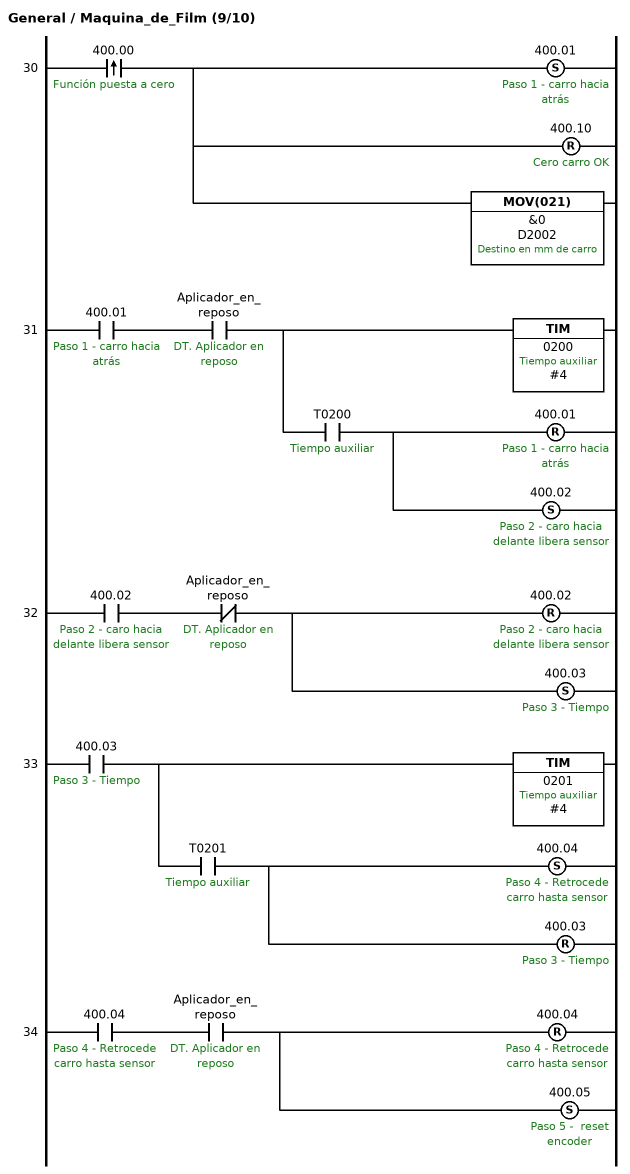
; [picture p24: General / Maquina_de_Film, rungs 30-34]
; rung 30
@LD 400.00  ; Función puesta a cero
SET 400.01  ; Paso 1 - carro hacia atrás
RSET 400.10  ; Cero carro OK
MOV(021) &0 D2002  ; Destino en mm de carro
; rung 31
LD 400.01  ; Paso 1 - carro hacia atrás
AND Aplicador_en_reposo  ; DT. Aplicador en reposo
TIM 0200 #4  ; Tiempo auxiliar
AND T0200  ; Tiempo auxiliar
RSET 400.01  ; Paso 1 - carro hacia atrás
SET 400.02  ; Paso 2 - caro hacia delante libera sensor
; rung 32
LD 400.02  ; Paso 2 - caro hacia delante libera sensor
ANDNOT Aplicador_en_reposo  ; DT. Aplicador en reposo
RSET 400.02  ; Paso 2 - caro hacia delante libera sensor
SET 400.03  ; Paso 3 - Tiempo
; rung 33
LD 400.03  ; Paso 3 - Tiempo
TIM 0201 #4  ; Tiempo auxiliar
AND T0201  ; Tiempo auxiliar
SET 400.04  ; Paso 4 - Retrocede carro hasta sensor
RSET 400.03  ; Paso 3 - Tiempo
; rung 34
LD 400.04  ; Paso 4 - Retrocede carro hasta sensor
AND Aplicador_en_reposo  ; DT. Aplicador en reposo
RSET 400.04  ; Paso 4 - Retrocede carro hasta sensor
SET 400.05  ; Paso 5 -  reset encoder

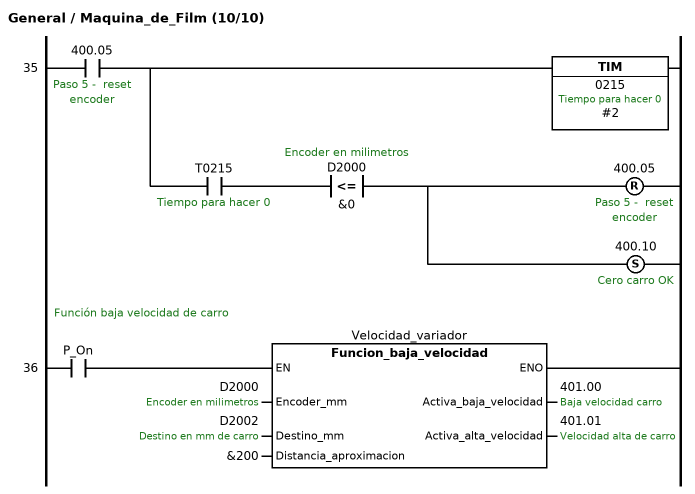
; rung 35
LD 400.05  ; Paso 5 -  reset encoder
TIM 0215 #2  ; Tiempo para hacer 0
AND T0215  ; Tiempo para hacer 0
AND<=SL(318) D2000 &0  ; Encoder en milimetros
RSET 400.05  ; Paso 5 -  reset encoder
SET 400.10  ; Cero carro OK
; rung 36: Función baja velocidad de carro
LD P_On
CALL Velocidad_variador : Funcion_baja_velocidad (Encoder_mm := D2000, Destino_mm := D2002, Distancia_aproximacion := &200, Activa_baja_velocidad => 401.00, Activa_alta_velocidad => 401.01)  ; Encoder en milimetros, Destino en mm de carro, Baja velocidad carro, Velocidad alta de carro

### Section Compuerta

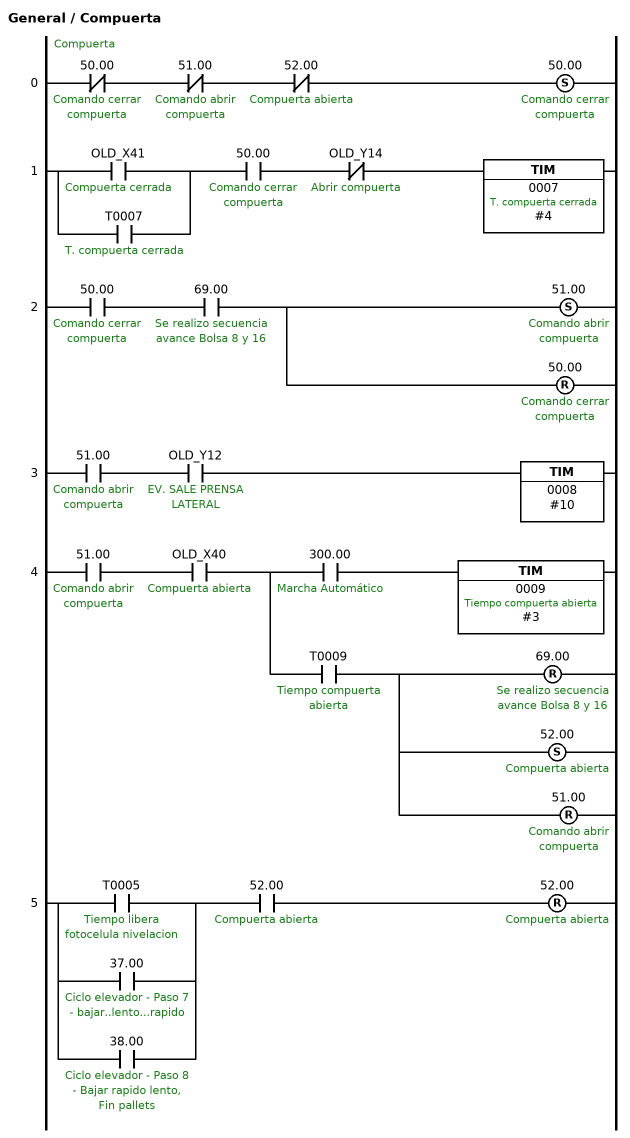
; rung 0: Compuerta
LDNOT 50.00  ; Comando cerrar compuerta
ANDNOT 51.00  ; Comando abrir compuerta
ANDNOT 52.00  ; Compuerta abierta
SET 50.00  ; Comando cerrar compuerta
; rung 1
LD OLD_X41  ; Compuerta cerrada
OR T0007  ; T. compuerta cerrada
AND 50.00  ; Comando cerrar compuerta
ANDNOT OLD_Y14  ; Abrir compuerta
TIM 0007 #4  ; T. compuerta cerrada
; rung 2
LD 50.00  ; Comando cerrar compuerta
AND 69.00  ; Se realizo secuencia avance Bolsa 8 y 16
SET 51.00  ; Comando abrir compuerta
RSET 50.00  ; Comando cerrar compuerta
; rung 3
LD 51.00  ; Comando abrir compuerta
AND OLD_Y12  ; EV. SALE PRENSA LATERAL
TIM 0008 #10
; rung 4
LD 51.00  ; Comando abrir compuerta
AND OLD_X40  ; Compuerta abierta
OUT TR0
AND 300.00  ; Marcha Automático
TIM 0009 #3  ; Tiempo compuerta abierta
LD TR0
AND T0009  ; Tiempo compuerta abierta
RSET 69.00  ; Se realizo secuencia avance Bolsa 8 y 16
SET 52.00  ; Compuerta abierta
RSET 51.00  ; Comando abrir compuerta
; rung 5
LD T0005  ; Tiempo libera fotocelula nivelacion
OR 37.00  ; Ciclo elevador - Paso 7 - bajar..lento...rapido
OR 38.00  ; Ciclo elevador - Paso 8 - Bajar rapido lento, Fin pallets
AND 52.00  ; Compuerta abierta
RSET 52.00  ; Compuerta abierta

### Section Carro_pala

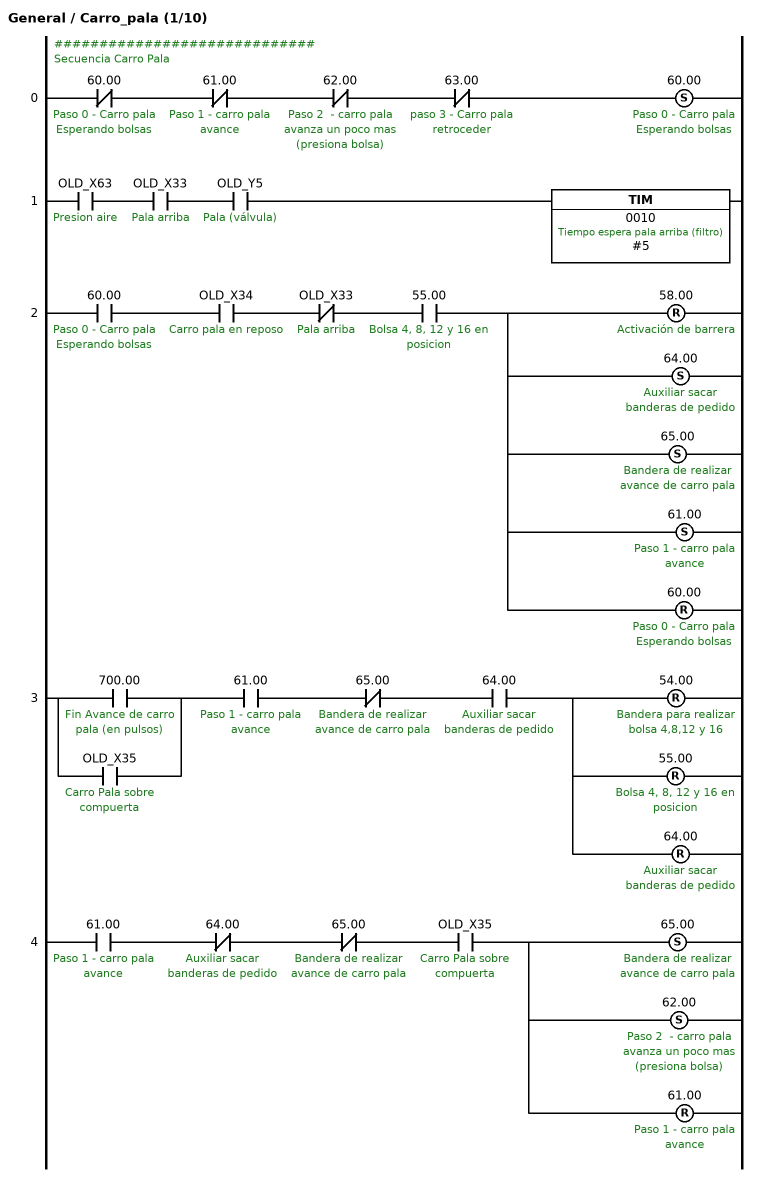
; rung 0: ############################# / Secuencia Carro Pala
LDNOT 60.00  ; Paso 0 - Carro pala Esperando bolsas
ANDNOT 61.00  ; Paso 1 - carro pala avance
ANDNOT 62.00  ; Paso 2  - carro pala avanza un poco mas (presiona bolsa)
ANDNOT 63.00  ; paso 3 - Carro pala retroceder
SET 60.00  ; Paso 0 - Carro pala Esperando bolsas
; rung 1
LD OLD_X63  ; Presion aire
AND OLD_X33  ; Pala arriba
AND OLD_Y5  ; Pala (válvula)
TIM 0010 #5  ; Tiempo espera pala arriba (filtro)
; rung 2
LD 60.00  ; Paso 0 - Carro pala Esperando bolsas
AND OLD_X34  ; Carro pala en reposo
ANDNOT OLD_X33  ; Pala arriba
AND 55.00  ; Bolsa 4, 8, 12 y 16 en posicion
RSET 58.00  ; Activación de barrera
SET 64.00  ; Auxiliar sacar banderas de pedido
SET 65.00  ; Bandera de realizar avance de carro pala
SET 61.00  ; Paso 1 - carro pala avance
RSET 60.00  ; Paso 0 - Carro pala Esperando bolsas
; rung 3
LD 700.00  ; Fin Avance de carro pala (en pulsos)
OR OLD_X35  ; Carro Pala sobre compuerta
AND 61.00  ; Paso 1 - carro pala avance
ANDNOT 65.00  ; Bandera de realizar avance de carro pala
AND 64.00  ; Auxiliar sacar banderas de pedido
RSET 54.00  ; Bandera para realizar bolsa 4,8,12 y 16
RSET 55.00  ; Bolsa 4, 8, 12 y 16 en posicion
RSET 64.00  ; Auxiliar sacar banderas de pedido
; rung 4
LD 61.00  ; Paso 1 - carro pala avance
ANDNOT 64.00  ; Auxiliar sacar banderas de pedido
ANDNOT 65.00  ; Bandera de realizar avance de carro pala
AND OLD_X35  ; Carro Pala sobre compuerta
SET 65.00  ; Bandera de realizar avance de carro pala
SET 62.00  ; Paso 2  - carro pala avanza un poco mas (presiona bolsa)
RSET 61.00  ; Paso 1 - carro pala avance

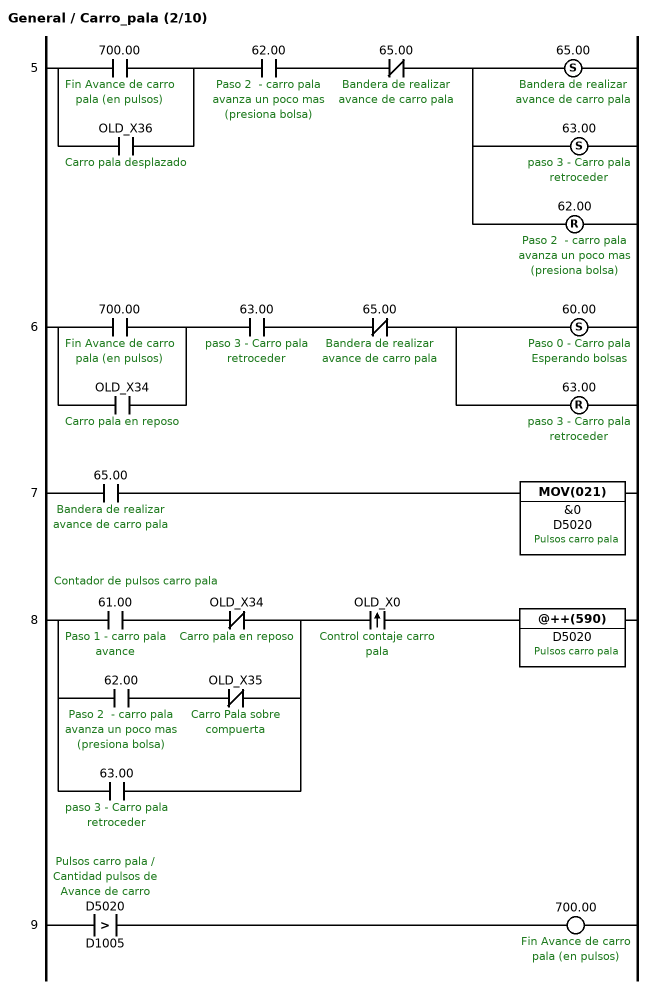
; rung 5
LD 700.00  ; Fin Avance de carro pala (en pulsos)
OR OLD_X36  ; Carro pala desplazado
AND 62.00  ; Paso 2  - carro pala avanza un poco mas (presiona bolsa)
ANDNOT 65.00  ; Bandera de realizar avance de carro pala
SET 65.00  ; Bandera de realizar avance de carro pala
SET 63.00  ; paso 3 - Carro pala retroceder
RSET 62.00  ; Paso 2  - carro pala avanza un poco mas (presiona bolsa)
; rung 6
LD 700.00  ; Fin Avance de carro pala (en pulsos)
OR OLD_X34  ; Carro pala en reposo
AND 63.00  ; paso 3 - Carro pala retroceder
ANDNOT 65.00  ; Bandera de realizar avance de carro pala
SET 60.00  ; Paso 0 - Carro pala Esperando bolsas
RSET 63.00  ; paso 3 - Carro pala retroceder
; rung 7
LD 65.00  ; Bandera de realizar avance de carro pala
MOV(021) &0 D5020  ; Pulsos carro pala
; rung 8: Contador de pulsos carro pala
LD 61.00  ; Paso 1 - carro pala avance
ANDNOT OLD_X34  ; Carro pala en reposo
LD 62.00  ; Paso 2  - carro pala avanza un poco mas (presiona bolsa)
ANDNOT OLD_X35  ; Carro Pala sobre compuerta
ORLD
OR 63.00  ; paso 3 - Carro pala retroceder
@AND OLD_X0  ; Control contaje carro pala
@++(590) D5020  ; Pulsos carro pala
; rung 9
LD>(320) D5020 D1005  ; Pulsos carro pala, Cantidad pulsos de Avance de carro
OUT 700.00  ; Fin Avance de carro pala (en pulsos)

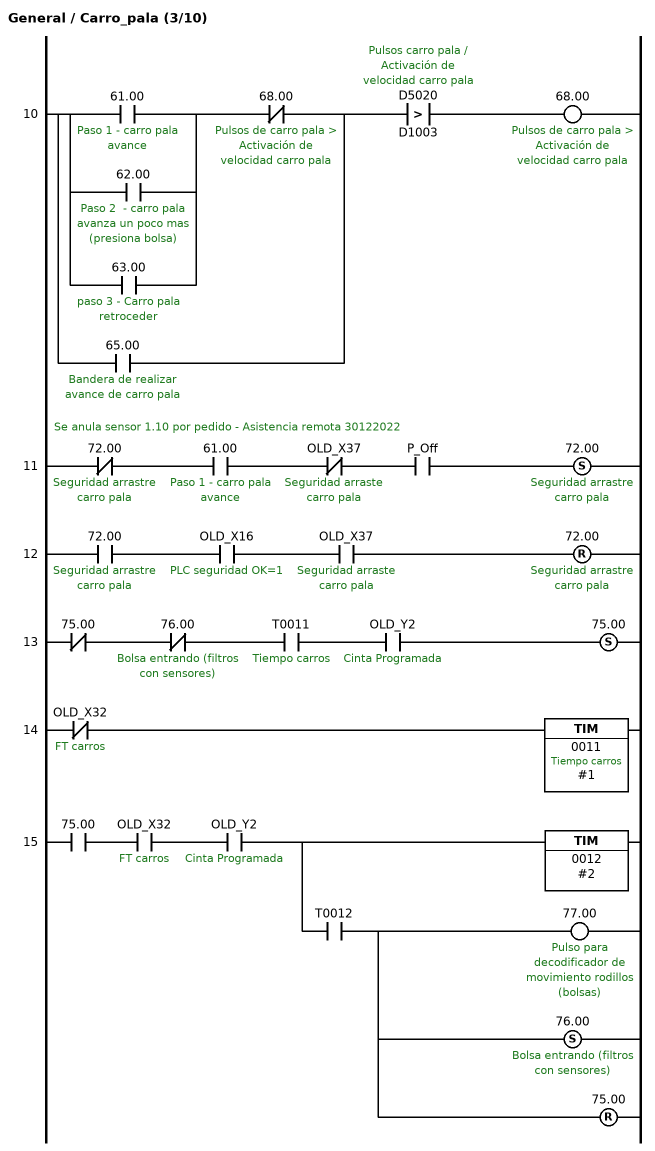
; rung 10
LD 61.00  ; Paso 1 - carro pala avance
OR 62.00  ; Paso 2  - carro pala avanza un poco mas (presiona bolsa)
OR 63.00  ; paso 3 - Carro pala retroceder
ANDNOT 68.00  ; Pulsos de carro pala > Activación de velocidad carro pala
OR 65.00  ; Bandera de realizar avance de carro pala
AND>L(321) D5020 D1003  ; Pulsos carro pala, Activación de velocidad carro pala
OUT 68.00  ; Pulsos de carro pala > Activación de velocidad carro pala
; rung 11: Se anula sensor 1.10 por pedido - Asistencia remota 30122022
LDNOT 72.00  ; Seguridad arrastre carro pala
AND 61.00  ; Paso 1 - carro pala avance
ANDNOT OLD_X37  ; Seguridad arraste carro pala
AND P_Off
SET 72.00  ; Seguridad arrastre carro pala
; rung 12
LD 72.00  ; Seguridad arrastre carro pala
AND OLD_X16  ; PLC seguridad OK=1
AND OLD_X37  ; Seguridad arraste carro pala
RSET 72.00  ; Seguridad arrastre carro pala
; rung 13
LDNOT 75.00
ANDNOT 76.00  ; Bolsa entrando (filtros con sensores)
AND T0011  ; Tiempo carros
AND OLD_Y2  ; Cinta Programada
SET 75.00
; rung 14
LDNOT OLD_X32  ; FT carros
TIM 0011 #1  ; Tiempo carros
; rung 15
LD 75.00
AND OLD_X32  ; FT carros
AND OLD_Y2  ; Cinta Programada
TIM 0012 #2  // Timer OK
AND T0012
OUT 77.00  ; Pulso para decodificador de movimiento rodillos (bolsas)
SET 76.00  ; Bolsa entrando (filtros con sensores)
RSET 75.00

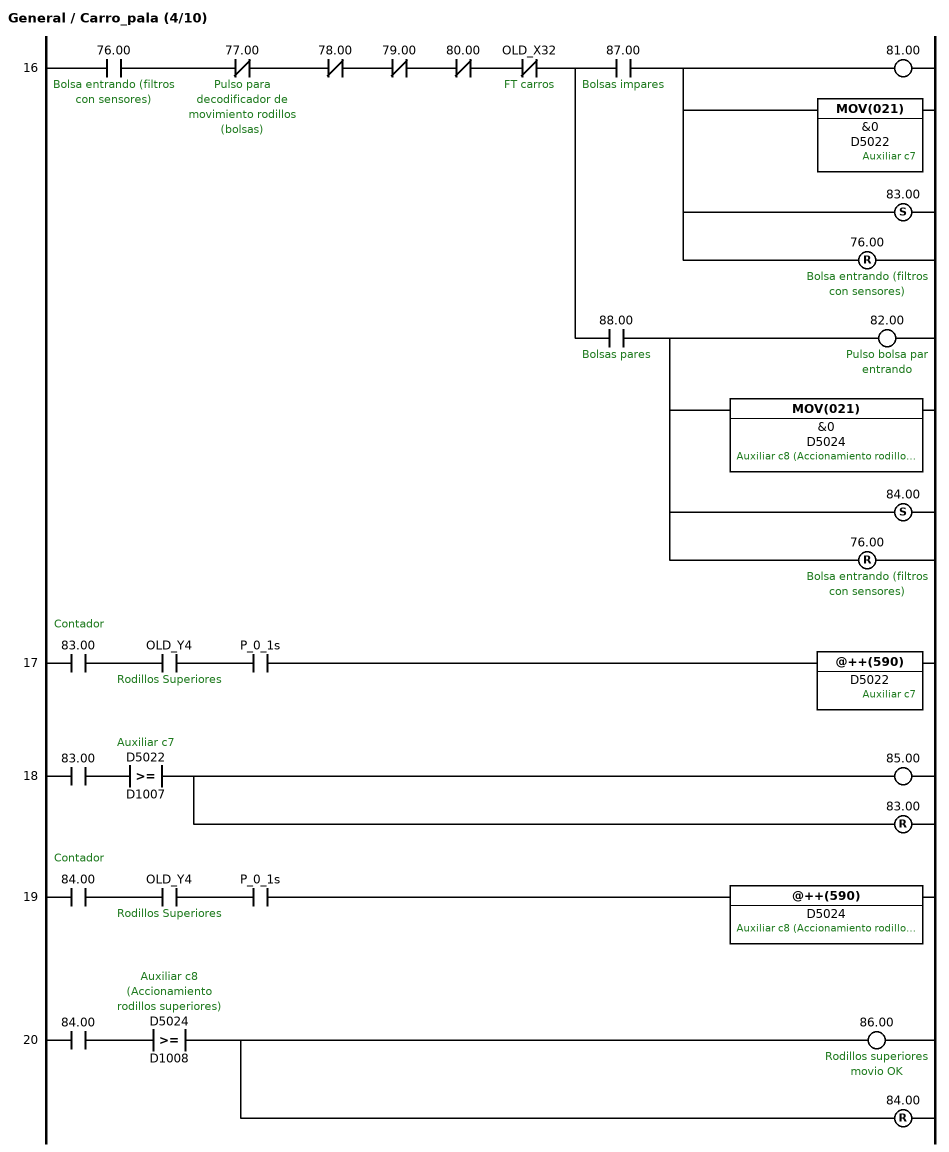
; rung 16
LD 76.00  ; Bolsa entrando (filtros con sensores)
ANDNOT 77.00  ; Pulso para decodificador de movimiento rodillos (bolsas)
ANDNOT 78.00
ANDNOT 79.00
ANDNOT 80.00
ANDNOT OLD_X32  ; FT carros
OUT TR0
AND 87.00  ; Bolsas impares
OUT 81.00
MOV(021) &0 D5022  ; Auxiliar c7
SET 83.00
RSET 76.00  ; Bolsa entrando (filtros con sensores)
LD TR0
AND 88.00  ; Bolsas pares
OUT 82.00  ; Pulso bolsa par entrando
MOV(021) &0 D5024  ; Auxiliar c8 (Accionamiento rodillos superiores)
SET 84.00
RSET 76.00  ; Bolsa entrando (filtros con sensores)
; rung 17: Contador
LD 83.00
AND OLD_Y4  ; Rodillos Superiores
AND P_0_1s
@++(590) D5022  ; Auxiliar c7
; rung 18
LD 83.00
AND>=(325) D5022 D1007  ; Auxiliar c7
OUT 85.00
RSET 83.00
; rung 19: Contador
LD 84.00
AND OLD_Y4  ; Rodillos Superiores
AND P_0_1s
@++(590) D5024  ; Auxiliar c8 (Accionamiento rodillos superiores)
; rung 20
LD 84.00
AND>=(325) D5024 D1008  ; Auxiliar c8 (Accionamiento rodillos superiores)
OUT 86.00  ; Rodillos superiores movio OK
RSET 84.00

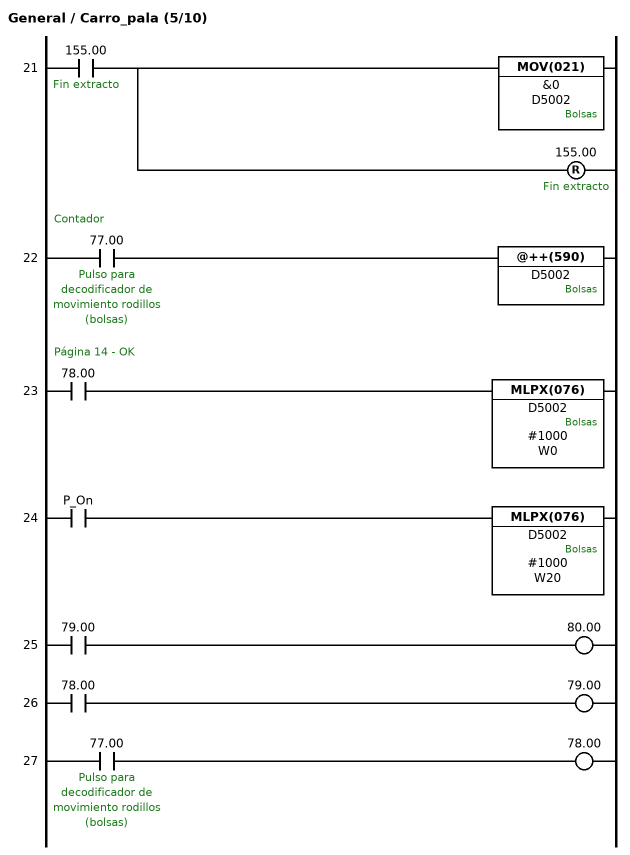
; rung 21
LD 155.00  ; Fin extracto
MOV(021) &0 D5002  ; Bolsas
RSET 155.00  ; Fin extracto
; rung 22: Contador
LD 77.00  ; Pulso para decodificador de movimiento rodillos (bolsas)
@++(590) D5002  ; Bolsas
; rung 23: Página 14 - OK
LD 78.00
MLPX(076) D5002 #1000 W0  ; Bolsas  // Decodificador tiempo de movimiento rodillos
; rung 24
LD P_On
MLPX(076) D5002 #1000 W20  ; Bolsas
; rung 25
LD 79.00
OUT 80.00
; rung 26
LD 78.00
OUT 79.00
; rung 27
LD 77.00  ; Pulso para decodificador de movimiento rodillos (bolsas)
OUT 78.00

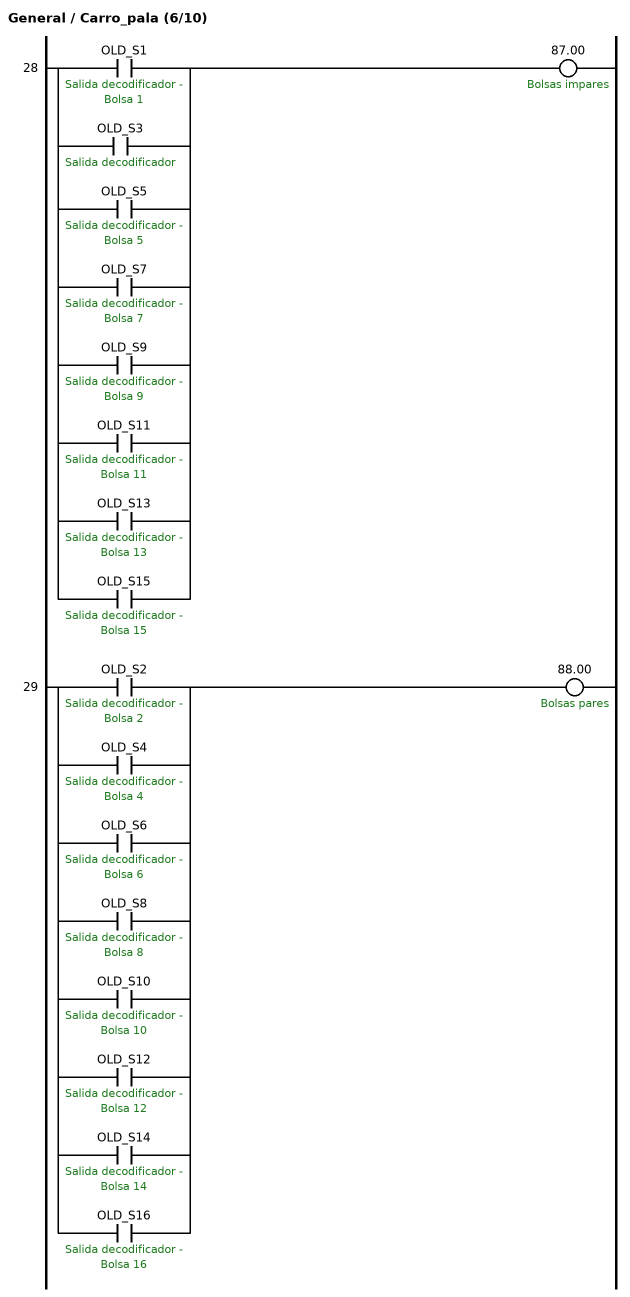
; rung 28
LD OLD_S1  ; Salida decodificador - Bolsa 1
OR OLD_S3  ; Salida decodificador
OR OLD_S5  ; Salida decodificador - Bolsa 5
OR OLD_S7  ; Salida decodificador - Bolsa 7
OR OLD_S9  ; Salida decodificador - Bolsa 9
OR OLD_S11  ; Salida decodificador - Bolsa 11
OR OLD_S13  ; Salida decodificador - Bolsa 13
OR OLD_S15  ; Salida decodificador - Bolsa 15
OUT 87.00  ; Bolsas impares
; rung 29
LD OLD_S2  ; Salida decodificador - Bolsa 2
OR OLD_S4  ; Salida decodificador - Bolsa 4
OR OLD_S6  ; Salida decodificador - Bolsa 6
OR OLD_S8  ; Salida decodificador - Bolsa 8
OR OLD_S10  ; Salida decodificador - Bolsa 10
OR OLD_S12  ; Salida decodificador - Bolsa 12
OR OLD_S14  ; Salida decodificador - Bolsa 14
OR OLD_S16  ; Salida decodificador - Bolsa 16
OUT 88.00  ; Bolsas pares

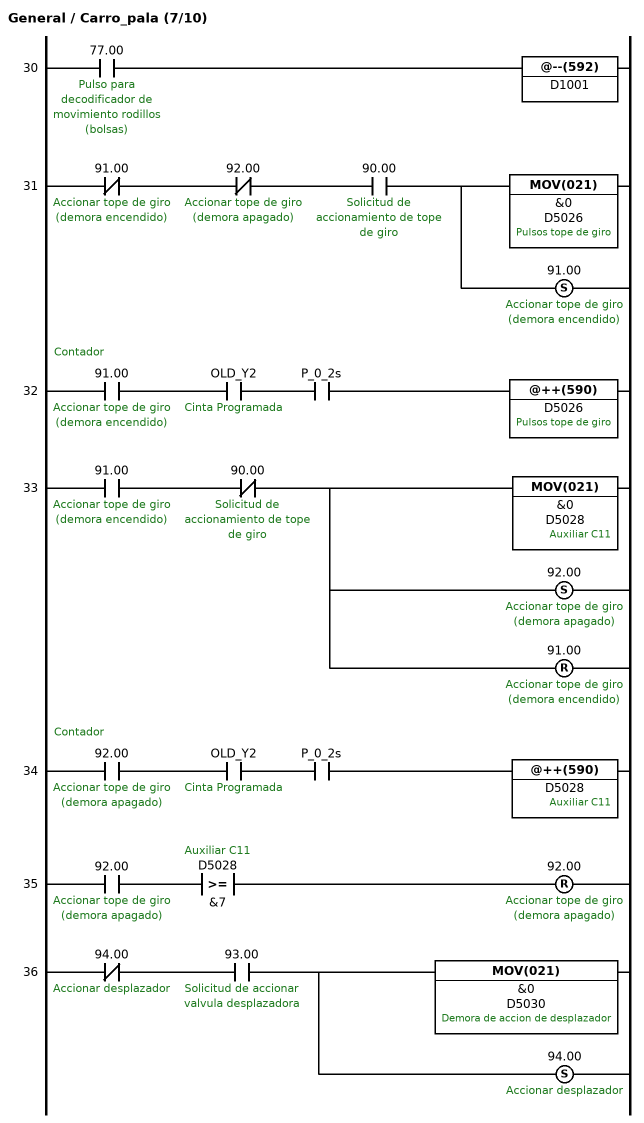
; rung 30
LD 77.00  ; Pulso para decodificador de movimiento rodillos (bolsas)
@--(592) D1001
; rung 31
LDNOT 91.00  ; Accionar tope de giro (demora encendido)
ANDNOT 92.00  ; Accionar tope de giro (demora apagado)
AND 90.00  ; Solicitud de accionamiento de tope de giro
MOV(021) &0 D5026  ; Pulsos tope de giro
SET 91.00  ; Accionar tope de giro (demora encendido)
; rung 32: Contador
LD 91.00  ; Accionar tope de giro (demora encendido)
AND OLD_Y2  ; Cinta Programada
AND P_0_2s
@++(590) D5026  ; Pulsos tope de giro
; rung 33
LD 91.00  ; Accionar tope de giro (demora encendido)
ANDNOT 90.00  ; Solicitud de accionamiento de tope de giro
MOV(021) &0 D5028  ; Auxiliar C11
SET 92.00  ; Accionar tope de giro (demora apagado)
RSET 91.00  ; Accionar tope de giro (demora encendido)
; rung 34: Contador
LD 92.00  ; Accionar tope de giro (demora apagado)
AND OLD_Y2  ; Cinta Programada
AND P_0_2s
@++(590) D5028  ; Auxiliar C11
; rung 35
LD 92.00  ; Accionar tope de giro (demora apagado)
AND>=(325) D5028 &7  ; Auxiliar C11
RSET 92.00  ; Accionar tope de giro (demora apagado)
; rung 36
LDNOT 94.00  ; Accionar desplazador
AND 93.00  ; Solicitud de accionar valvula desplazadora
MOV(021) &0 D5030  ; Demora de accion de desplazador
SET 94.00  ; Accionar desplazador

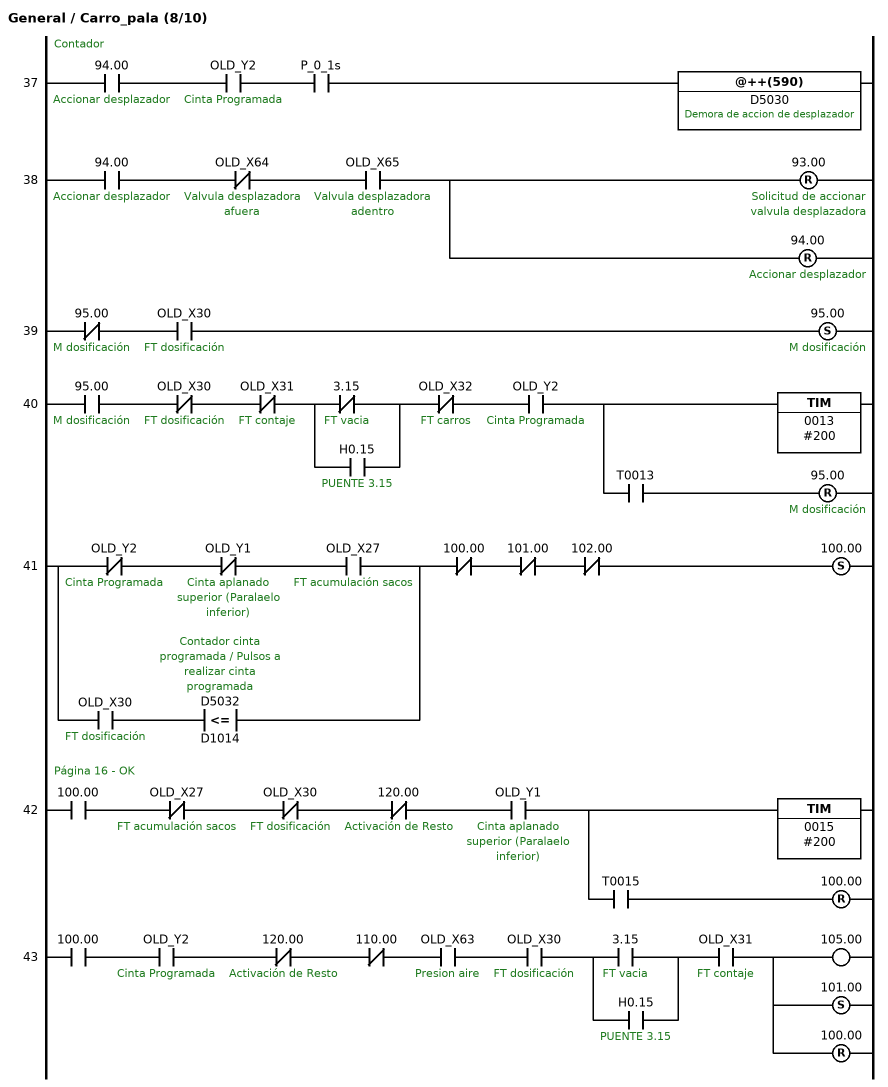
; rung 37: Contador
LD 94.00  ; Accionar desplazador
AND OLD_Y2  ; Cinta Programada
AND P_0_1s
@++(590) D5030  ; Demora de accion de desplazador
; rung 38
LD 94.00  ; Accionar desplazador
ANDNOT OLD_X64  ; Valvula desplazadora afuera
AND OLD_X65  ; Valvula desplazadora adentro
RSET 93.00  ; Solicitud de accionar valvula desplazadora
RSET 94.00  ; Accionar desplazador
; rung 39
LDNOT 95.00  ; M dosificación
AND OLD_X30  ; FT dosificación
SET 95.00  ; M dosificación
; rung 40
LD 95.00  ; M dosificación
ANDNOT OLD_X30  ; FT dosificación
ANDNOT OLD_X31  ; FT contaje
LDNOT 3.15  ; FT vacia
OR H0.15  ; PUENTE 3.15
ANDLD
ANDNOT OLD_X32  ; FT carros
AND OLD_Y2  ; Cinta Programada
TIM 0013 #200
AND T0013
RSET 95.00  ; M dosificación
; rung 41
LDNOT OLD_Y2  ; Cinta Programada
ANDNOT OLD_Y1  ; Cinta aplanado superior (Paralaelo inferior)
AND OLD_X27  ; FT acumulación sacos
LD OLD_X30  ; FT dosificación
AND<=(315) D5032 D1014  ; Contador cinta programada, Pulsos a realizar cinta programada
ORLD
ANDNOT 100.00
ANDNOT 101.00
ANDNOT 102.00
SET 100.00
; rung 42: Página 16 - OK
LD 100.00
ANDNOT OLD_X27  ; FT acumulación sacos
ANDNOT OLD_X30  ; FT dosificación
ANDNOT 120.00  ; Activación de Resto
AND OLD_Y1  ; Cinta aplanado superior (Paralaelo inferior)
TIM 0015 #200
AND T0015
RSET 100.00
; rung 43
LD 100.00
AND OLD_Y2  ; Cinta Programada
ANDNOT 120.00  ; Activación de Resto
ANDNOT 110.00
AND OLD_X63  ; Presion aire
AND OLD_X30  ; FT dosificación
LD 3.15  ; FT vacia
OR H0.15  ; PUENTE 3.15
ANDLD
AND OLD_X31  ; FT contaje
OUT 105.00
SET 101.00
RSET 100.00

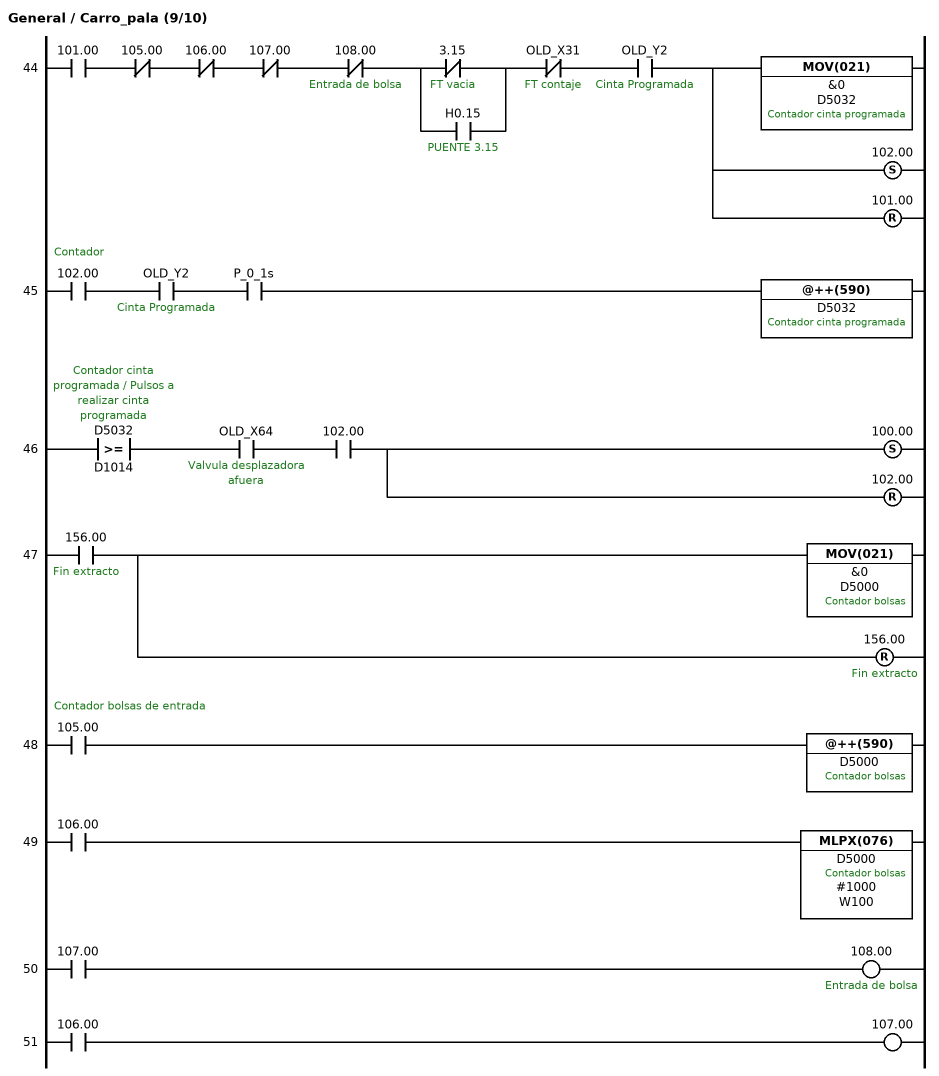
; rung 44
LD 101.00
ANDNOT 105.00
ANDNOT 106.00
ANDNOT 107.00
ANDNOT 108.00  ; Entrada de bolsa
LDNOT 3.15  ; FT vacia
OR H0.15  ; PUENTE 3.15
ANDLD
ANDNOT OLD_X31  ; FT contaje
AND OLD_Y2  ; Cinta Programada
MOV(021) &0 D5032  ; Contador cinta programada
SET 102.00
RSET 101.00
; rung 45: Contador
LD 102.00
AND OLD_Y2  ; Cinta Programada
AND P_0_1s
@++(590) D5032  ; Contador cinta programada
; rung 46
LD>=(325) D5032 D1014  ; Contador cinta programada, Pulsos a realizar cinta programada
AND OLD_X64  ; Valvula desplazadora afuera
AND 102.00
SET 100.00
RSET 102.00
; rung 47
LD 156.00  ; Fin extracto
MOV(021) &0 D5000  ; Contador bolsas
RSET 156.00  ; Fin extracto
; rung 48: Contador bolsas de entrada
LD 105.00
@++(590) D5000  ; Contador bolsas
; rung 49
LD 106.00
MLPX(076) D5000 #1000 W100  ; Contador bolsas  // Decodificador para movimientos, tiempos de pala lateral, valvula giradora
; rung 50
LD 107.00
OUT 108.00  ; Entrada de bolsa
; rung 51
LD 106.00
OUT 107.00

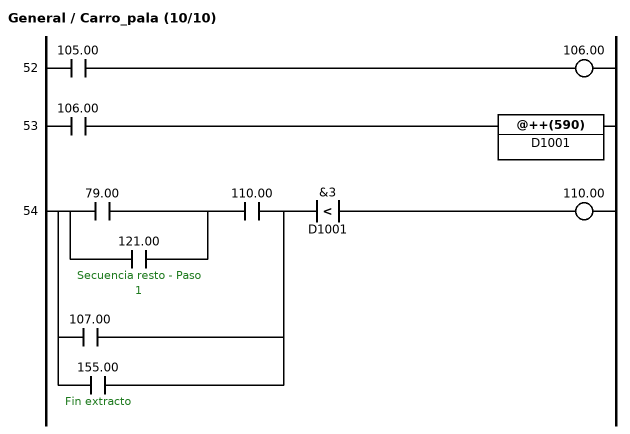
; rung 52
LD 105.00
OUT 106.00
; rung 53
LD 106.00
@++(590) D1001
; rung 54
LD 79.00
OR 121.00  ; Secuencia resto - Paso 1
AND 110.00
OR 107.00
OR 155.00  ; Fin extracto
AND<(310) &3 D1001
OUT 110.00

### Section Resto

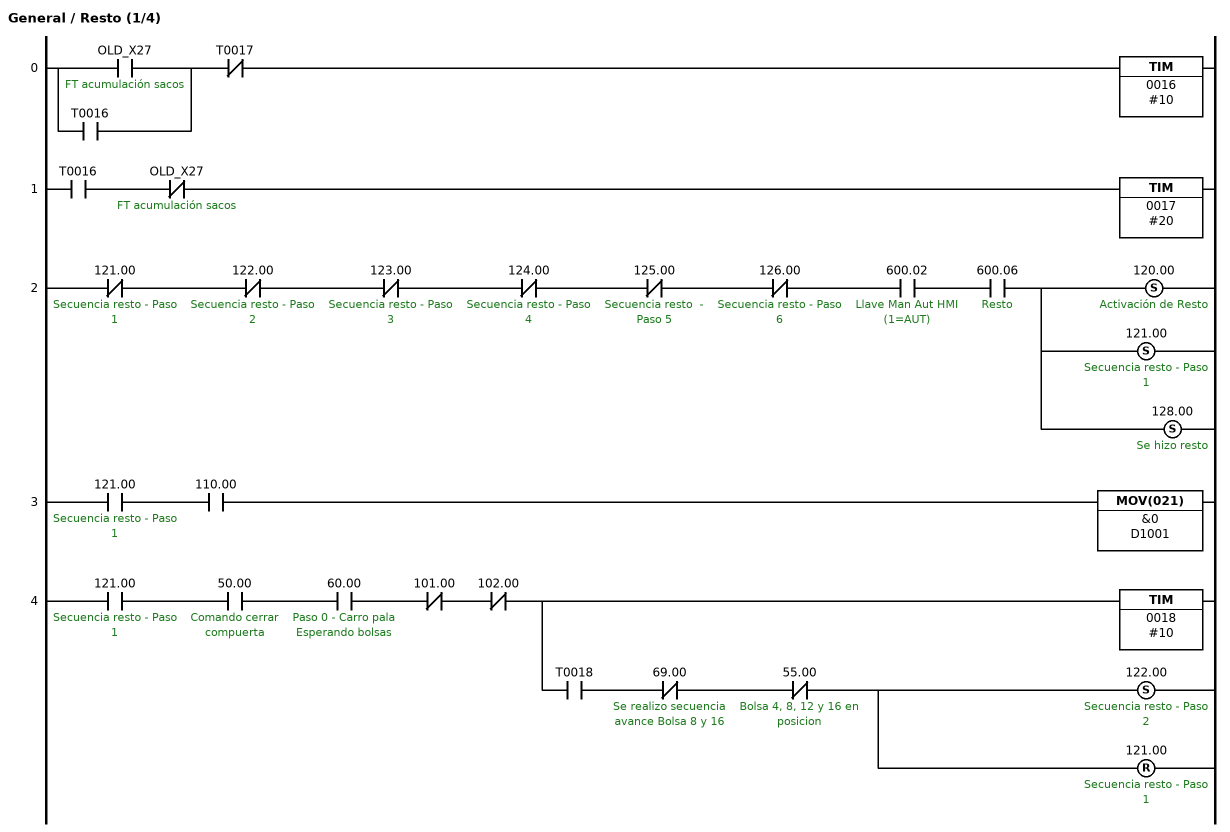
; rung 0
LD OLD_X27  ; FT acumulación sacos
OR T0016
ANDNOT T0017
TIM 0016 #10
; rung 1
LD T0016
ANDNOT OLD_X27  ; FT acumulación sacos
TIM 0017 #20
; rung 2
LDNOT 121.00  ; Secuencia resto - Paso 1
ANDNOT 122.00  ; Secuencia resto - Paso 2
ANDNOT 123.00  ; Secuencia resto - Paso 3
ANDNOT 124.00  ; Secuencia resto - Paso 4
ANDNOT 125.00  ; Secuencia resto  - Paso 5
ANDNOT 126.00  ; Secuencia resto - Paso 6
AND 600.02  ; Llave Man Aut HMI (1=AUT)
AND 600.06  ; Resto
SET 120.00  ; Activación de Resto
SET 121.00  ; Secuencia resto - Paso 1
SET 128.00  ; Se hizo resto
; rung 3
LD 121.00  ; Secuencia resto - Paso 1
AND 110.00
MOV(021) &0 D1001
; rung 4
LD 121.00  ; Secuencia resto - Paso 1
AND 50.00  ; Comando cerrar compuerta
AND 60.00  ; Paso 0 - Carro pala Esperando bolsas
ANDNOT 101.00
ANDNOT 102.00
TIM 0018 #10
AND T0018
ANDNOT 69.00  ; Se realizo secuencia avance Bolsa 8 y 16
ANDNOT 55.00  ; Bolsa 4, 8, 12 y 16 en posicion
SET 122.00  ; Secuencia resto - Paso 2
RSET 121.00  ; Secuencia resto - Paso 1

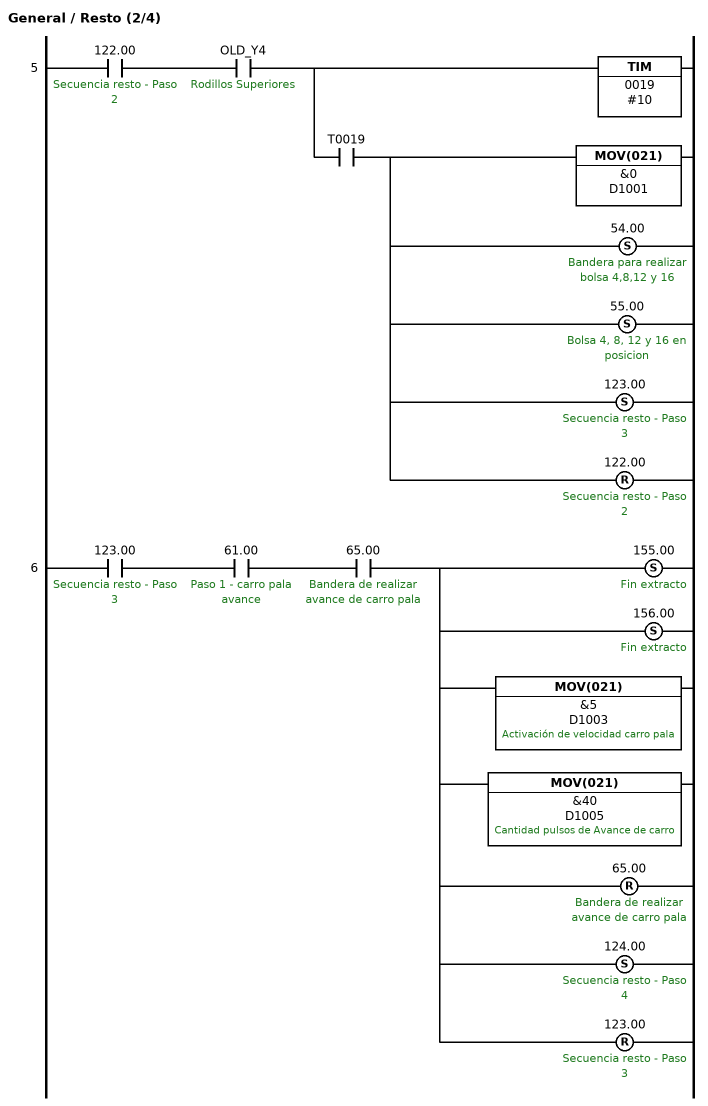
; rung 5
LD 122.00  ; Secuencia resto - Paso 2
AND OLD_Y4  ; Rodillos Superiores
TIM 0019 #10
AND T0019
MOV(021) &0 D1001
SET 54.00  ; Bandera para realizar bolsa 4,8,12 y 16
SET 55.00  ; Bolsa 4, 8, 12 y 16 en posicion
SET 123.00  ; Secuencia resto - Paso 3
RSET 122.00  ; Secuencia resto - Paso 2
; rung 6
LD 123.00  ; Secuencia resto - Paso 3
AND 61.00  ; Paso 1 - carro pala avance
AND 65.00  ; Bandera de realizar avance de carro pala
SET 155.00  ; Fin extracto
SET 156.00  ; Fin extracto
MOV(021) &5 D1003  ; Activación de velocidad carro pala
MOV(021) &40 D1005  ; Cantidad pulsos de Avance de carro
RSET 65.00  ; Bandera de realizar avance de carro pala
SET 124.00  ; Secuencia resto - Paso 4
RSET 123.00  ; Secuencia resto - Paso 3

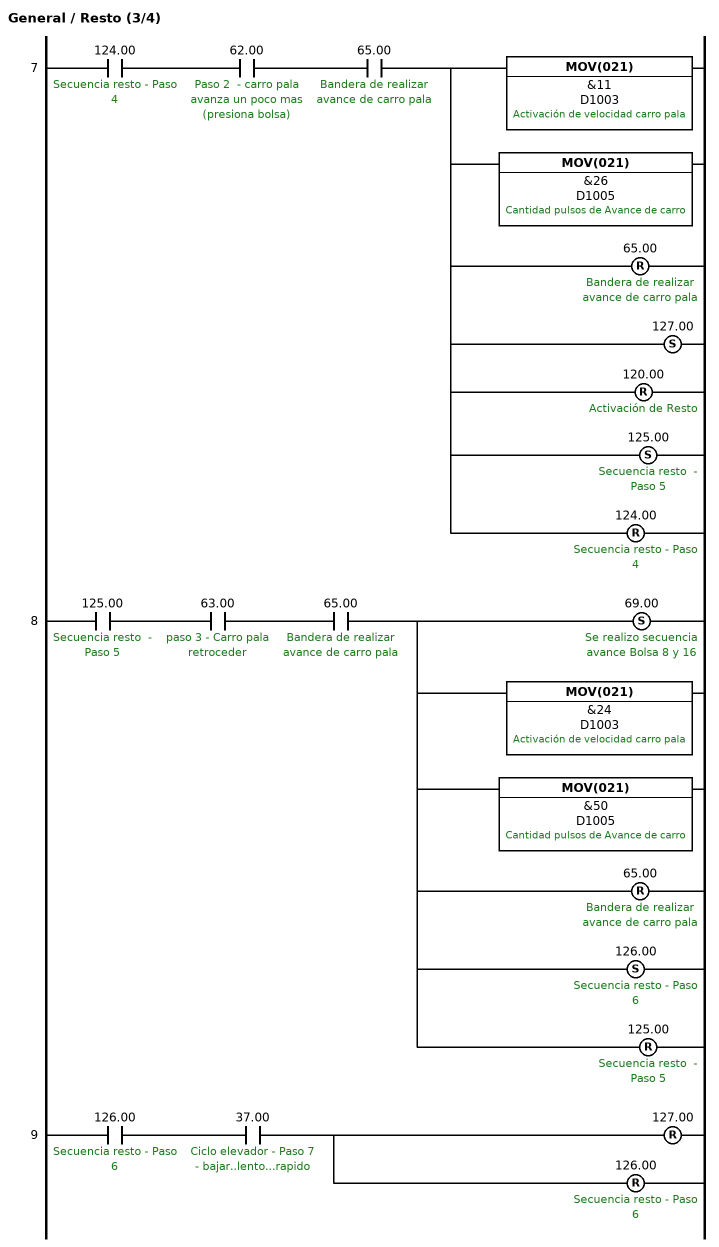
; rung 7
LD 124.00  ; Secuencia resto - Paso 4
AND 62.00  ; Paso 2  - carro pala avanza un poco mas (presiona bolsa)
AND 65.00  ; Bandera de realizar avance de carro pala
MOV(021) &11 D1003  ; Activación de velocidad carro pala
MOV(021) &26 D1005  ; Cantidad pulsos de Avance de carro
RSET 65.00  ; Bandera de realizar avance de carro pala
SET 127.00
RSET 120.00  ; Activación de Resto
SET 125.00  ; Secuencia resto  - Paso 5
RSET 124.00  ; Secuencia resto - Paso 4
; rung 8
LD 125.00  ; Secuencia resto  - Paso 5
AND 63.00  ; paso 3 - Carro pala retroceder
AND 65.00  ; Bandera de realizar avance de carro pala
SET 69.00  ; Se realizo secuencia avance Bolsa 8 y 16
MOV(021) &24 D1003  ; Activación de velocidad carro pala
MOV(021) &50 D1005  ; Cantidad pulsos de Avance de carro
RSET 65.00  ; Bandera de realizar avance de carro pala
SET 126.00  ; Secuencia resto - Paso 6
RSET 125.00  ; Secuencia resto  - Paso 5
; rung 9
LD 126.00  ; Secuencia resto - Paso 6
AND 37.00  ; Ciclo elevador - Paso 7 - bajar..lento...rapido
RSET 127.00
RSET 126.00  ; Secuencia resto - Paso 6

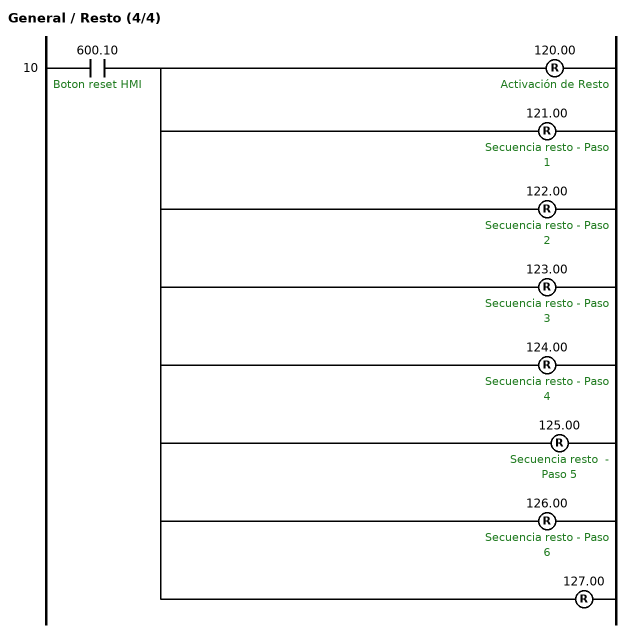
; rung 10
LD 600.10  ; Boton reset HMI
RSET 120.00  ; Activación de Resto
RSET 121.00  ; Secuencia resto - Paso 1
RSET 122.00  ; Secuencia resto - Paso 2
RSET 123.00  ; Secuencia resto - Paso 3
RSET 124.00  ; Secuencia resto - Paso 4
RSET 125.00  ; Secuencia resto  - Paso 5
RSET 126.00  ; Secuencia resto - Paso 6
RSET 127.00

### Section Secuencia_entrada_bolsa

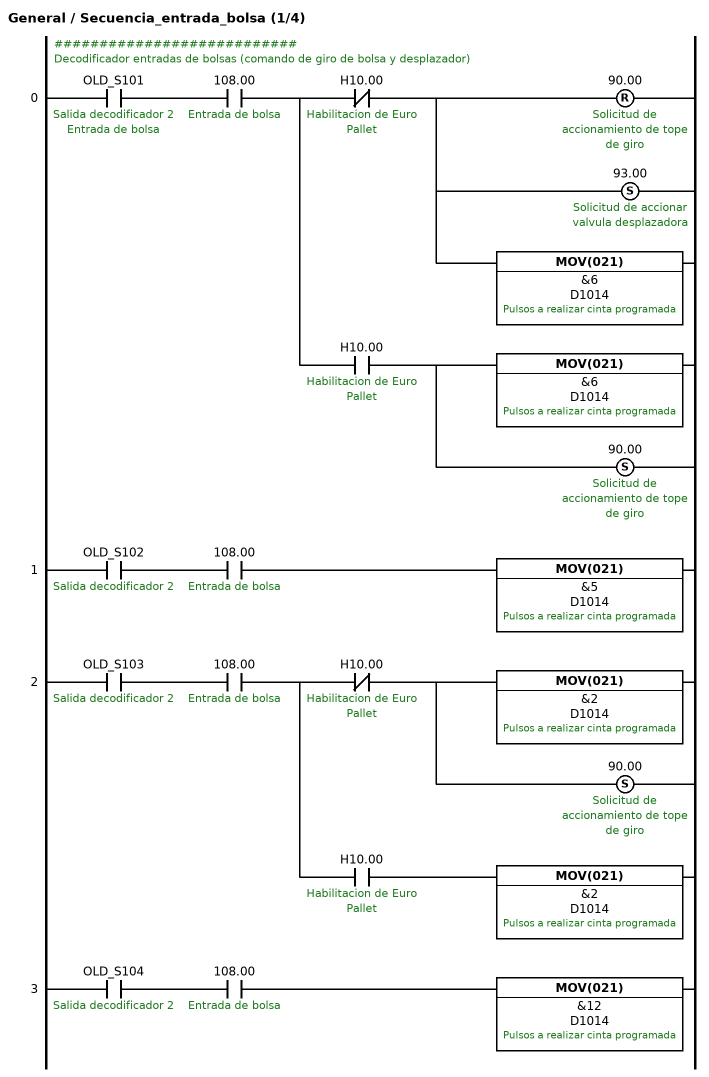
; rung 0: ########################### / Decodificador entradas de bolsas (comando de giro de bolsa y desplazador)
LD OLD_S101  ; Salida decodificador 2 Entrada de bolsa
AND 108.00  ; Entrada de bolsa
OUT TR0
ANDNOT H10.00  ; Habilitacion de Euro Pallet
RSET 90.00  ; Solicitud de accionamiento de tope de giro
SET 93.00  ; Solicitud de accionar valvula desplazadora
MOV(021) &6 D1014  ; Pulsos a realizar cinta programada
LD TR0
AND H10.00  ; Habilitacion de Euro Pallet
MOV(021) &6 D1014  ; Pulsos a realizar cinta programada
SET 90.00  ; Solicitud de accionamiento de tope de giro
; rung 1
LD OLD_S102  ; Salida decodificador 2
AND 108.00  ; Entrada de bolsa
MOV(021) &5 D1014  ; Pulsos a realizar cinta programada
; rung 2
LD OLD_S103  ; Salida decodificador 2
AND 108.00  ; Entrada de bolsa
OUT TR0
ANDNOT H10.00  ; Habilitacion de Euro Pallet
MOV(021) &2 D1014  ; Pulsos a realizar cinta programada
SET 90.00  ; Solicitud de accionamiento de tope de giro
LD TR0
AND H10.00  ; Habilitacion de Euro Pallet
MOV(021) &2 D1014  ; Pulsos a realizar cinta programada
; rung 3
LD OLD_S104  ; Salida decodificador 2
AND 108.00  ; Entrada de bolsa
MOV(021) &12 D1014  ; Pulsos a realizar cinta programada

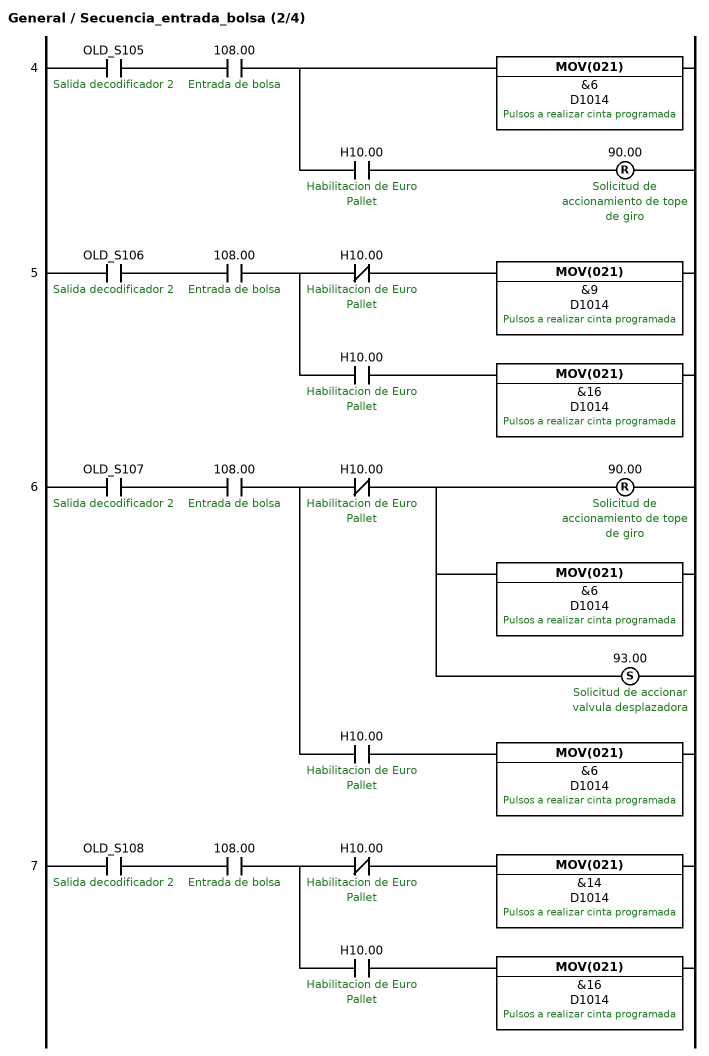
; rung 4
LD OLD_S105  ; Salida decodificador 2
AND 108.00  ; Entrada de bolsa
MOV(021) &6 D1014  ; Pulsos a realizar cinta programada
AND H10.00  ; Habilitacion de Euro Pallet
RSET 90.00  ; Solicitud de accionamiento de tope de giro
; rung 5
LD OLD_S106  ; Salida decodificador 2
AND 108.00  ; Entrada de bolsa
OUT TR0
ANDNOT H10.00  ; Habilitacion de Euro Pallet
MOV(021) &9 D1014  ; Pulsos a realizar cinta programada
LD TR0
AND H10.00  ; Habilitacion de Euro Pallet
MOV(021) &16 D1014  ; Pulsos a realizar cinta programada
; rung 6
LD OLD_S107  ; Salida decodificador 2
AND 108.00  ; Entrada de bolsa
OUT TR0
ANDNOT H10.00  ; Habilitacion de Euro Pallet
RSET 90.00  ; Solicitud de accionamiento de tope de giro
MOV(021) &6 D1014  ; Pulsos a realizar cinta programada
SET 93.00  ; Solicitud de accionar valvula desplazadora
LD TR0
AND H10.00  ; Habilitacion de Euro Pallet
MOV(021) &6 D1014  ; Pulsos a realizar cinta programada
; rung 7
LD OLD_S108  ; Salida decodificador 2
AND 108.00  ; Entrada de bolsa
OUT TR0
ANDNOT H10.00  ; Habilitacion de Euro Pallet
MOV(021) &14 D1014  ; Pulsos a realizar cinta programada
LD TR0
AND H10.00  ; Habilitacion de Euro Pallet
MOV(021) &16 D1014  ; Pulsos a realizar cinta programada

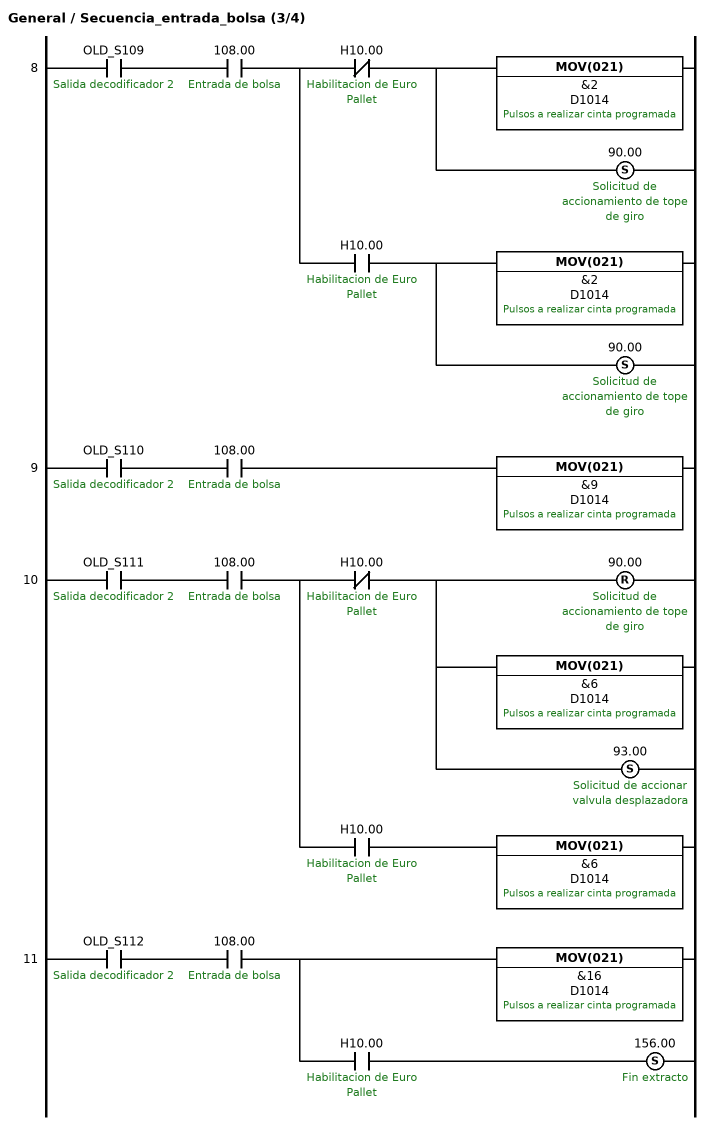
; rung 8
LD OLD_S109  ; Salida decodificador 2
AND 108.00  ; Entrada de bolsa
OUT TR0
ANDNOT H10.00  ; Habilitacion de Euro Pallet
MOV(021) &2 D1014  ; Pulsos a realizar cinta programada
SET 90.00  ; Solicitud de accionamiento de tope de giro
LD TR0
AND H10.00  ; Habilitacion de Euro Pallet
MOV(021) &2 D1014  ; Pulsos a realizar cinta programada
SET 90.00  ; Solicitud de accionamiento de tope de giro
; rung 9
LD OLD_S110  ; Salida decodificador 2
AND 108.00  ; Entrada de bolsa
MOV(021) &9 D1014  ; Pulsos a realizar cinta programada
; rung 10
LD OLD_S111  ; Salida decodificador 2
AND 108.00  ; Entrada de bolsa
OUT TR0
ANDNOT H10.00  ; Habilitacion de Euro Pallet
RSET 90.00  ; Solicitud de accionamiento de tope de giro
MOV(021) &6 D1014  ; Pulsos a realizar cinta programada
SET 93.00  ; Solicitud de accionar valvula desplazadora
LD TR0
AND H10.00  ; Habilitacion de Euro Pallet
MOV(021) &6 D1014  ; Pulsos a realizar cinta programada
; rung 11
LD OLD_S112  ; Salida decodificador 2
AND 108.00  ; Entrada de bolsa
MOV(021) &16 D1014  ; Pulsos a realizar cinta programada
AND H10.00  ; Habilitacion de Euro Pallet
SET 156.00  ; Fin extracto

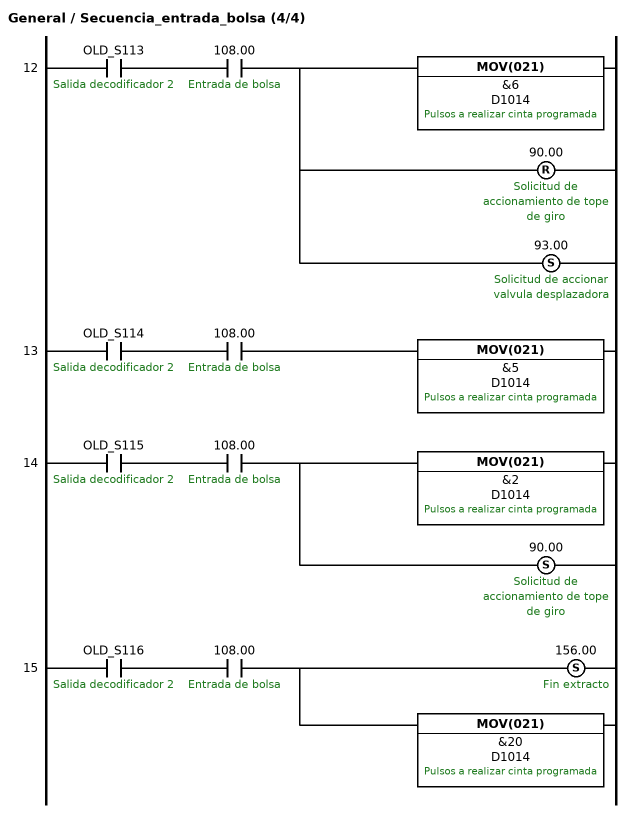
; rung 12
LD OLD_S113  ; Salida decodificador 2
AND 108.00  ; Entrada de bolsa
MOV(021) &6 D1014  ; Pulsos a realizar cinta programada
RSET 90.00  ; Solicitud de accionamiento de tope de giro
SET 93.00  ; Solicitud de accionar valvula desplazadora
; rung 13
LD OLD_S114  ; Salida decodificador 2
AND 108.00  ; Entrada de bolsa
MOV(021) &5 D1014  ; Pulsos a realizar cinta programada
; rung 14
LD OLD_S115  ; Salida decodificador 2
AND 108.00  ; Entrada de bolsa
MOV(021) &2 D1014  ; Pulsos a realizar cinta programada
SET 90.00  ; Solicitud de accionamiento de tope de giro
; rung 15
LD OLD_S116  ; Salida decodificador 2
AND 108.00  ; Entrada de bolsa
SET 156.00  ; Fin extracto
MOV(021) &20 D1014  ; Pulsos a realizar cinta programada

### Section Secuencia_rodillos_Pala

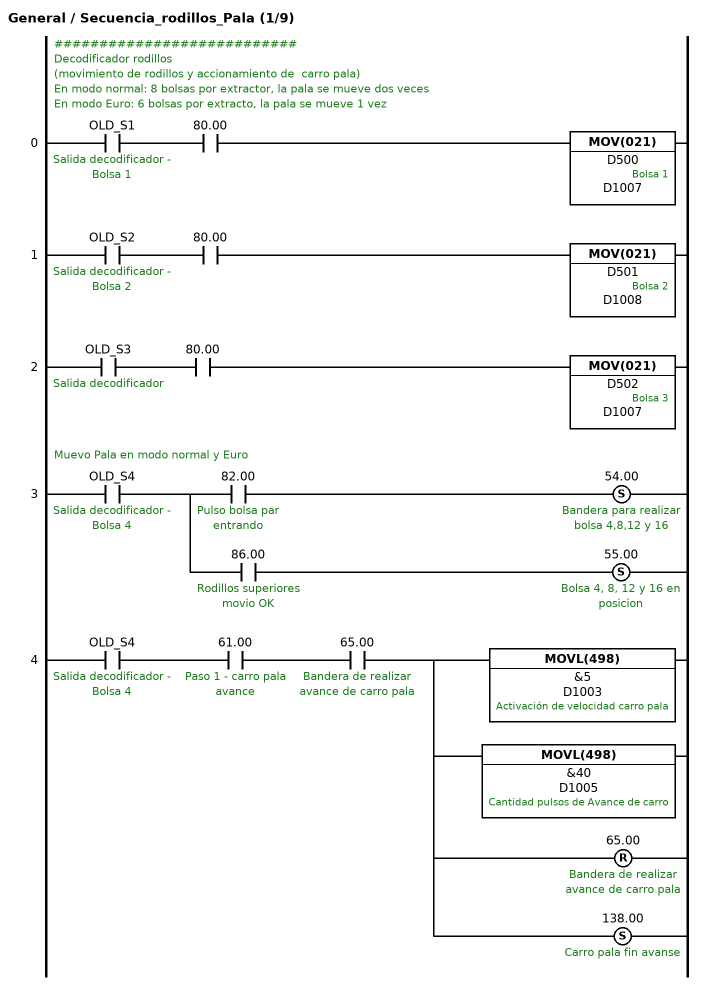
; rung 0: ########################### / Decodificador rodillos / (movimiento de rodillos y accionamiento de  carro pala) / En modo normal: 8 bolsas por extractor, la pala se mueve dos veces / En modo Euro: 6 bolsas por extracto, la pala se mueve 1 vez
LD OLD_S1  ; Salida decodificador - Bolsa 1
AND 80.00
MOV(021) D500 D1007  ; Bolsa 1
; rung 1
LD OLD_S2  ; Salida decodificador - Bolsa 2
AND 80.00
MOV(021) D501 D1008  ; Bolsa 2
; rung 2
LD OLD_S3  ; Salida decodificador
AND 80.00
MOV(021) D502 D1007  ; Bolsa 3
; rung 3: Muevo Pala en modo normal y Euro
LD OLD_S4  ; Salida decodificador - Bolsa 4
OUT TR0
AND 82.00  ; Pulso bolsa par entrando
SET 54.00  ; Bandera para realizar bolsa 4,8,12 y 16
LD TR0
AND 86.00  ; Rodillos superiores movio OK
SET 55.00  ; Bolsa 4, 8, 12 y 16 en posicion
; rung 4
LD OLD_S4  ; Salida decodificador - Bolsa 4
AND 61.00  ; Paso 1 - carro pala avance
AND 65.00  ; Bandera de realizar avance de carro pala
MOVL(498) &5 D1003  ; Activación de velocidad carro pala
MOVL(498) &40 D1005  ; Cantidad pulsos de Avance de carro
RSET 65.00  ; Bandera de realizar avance de carro pala
SET 138.00  ; Carro pala fin avanse

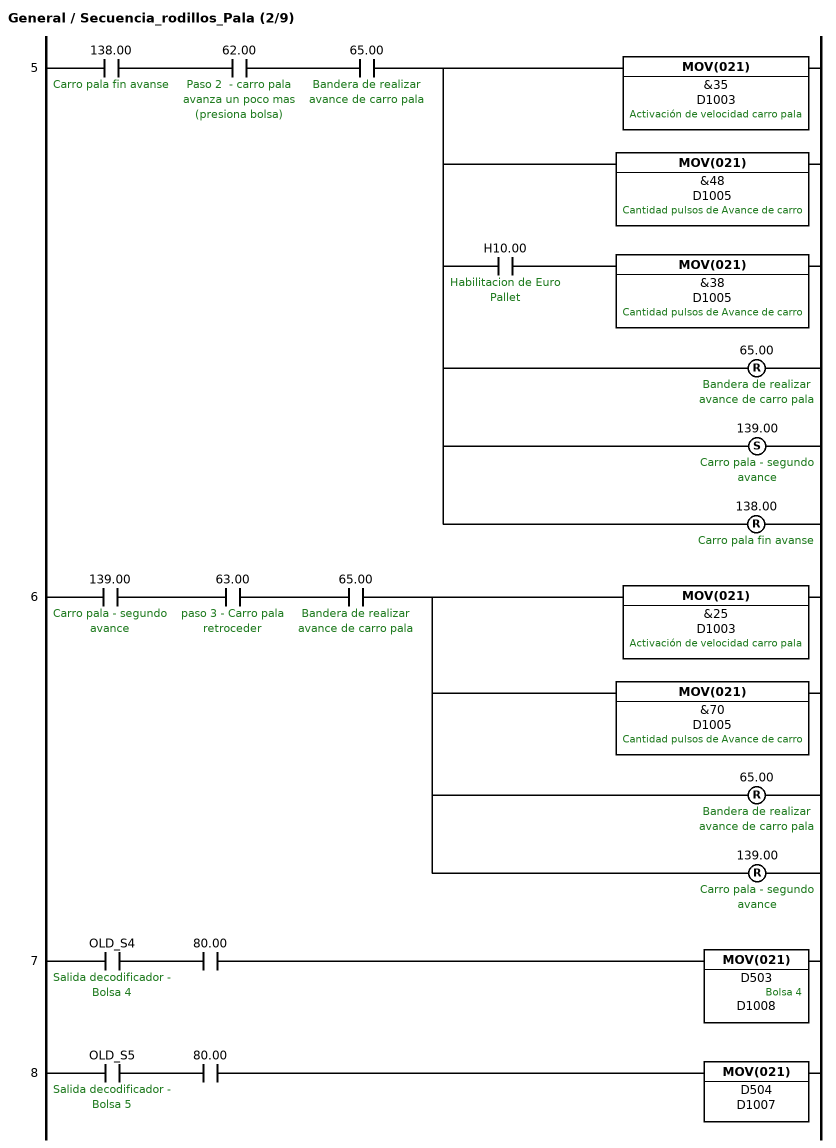
; rung 5
LD 138.00  ; Carro pala fin avanse
AND 62.00  ; Paso 2  - carro pala avanza un poco mas (presiona bolsa)
AND 65.00  ; Bandera de realizar avance de carro pala
OUT TR0
MOV(021) &35 D1003  ; Activación de velocidad carro pala
MOV(021) &48 D1005  ; Cantidad pulsos de Avance de carro
AND H10.00  ; Habilitacion de Euro Pallet
MOV(021) &38 D1005  ; Cantidad pulsos de Avance de carro
LD TR0
RSET 65.00  ; Bandera de realizar avance de carro pala
SET 139.00  ; Carro pala - segundo avance
RSET 138.00  ; Carro pala fin avanse
; rung 6
LD 139.00  ; Carro pala - segundo avance
AND 63.00  ; paso 3 - Carro pala retroceder
AND 65.00  ; Bandera de realizar avance de carro pala
MOV(021) &25 D1003  ; Activación de velocidad carro pala
MOV(021) &70 D1005  ; Cantidad pulsos de Avance de carro
RSET 65.00  ; Bandera de realizar avance de carro pala
RSET 139.00  ; Carro pala - segundo avance
; rung 7
LD OLD_S4  ; Salida decodificador - Bolsa 4
AND 80.00
MOV(021) D503 D1008  ; Bolsa 4  // Original valor &8
; rung 8
LD OLD_S5  ; Salida decodificador - Bolsa 5
AND 80.00
MOV(021) D504 D1007

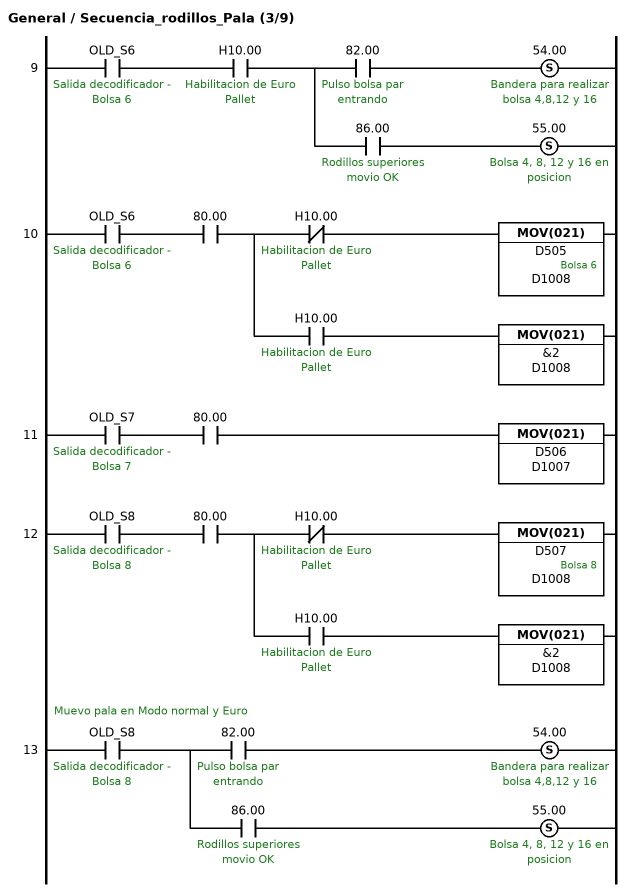
; rung 9
LD OLD_S6  ; Salida decodificador - Bolsa 6
AND H10.00  ; Habilitacion de Euro Pallet
OUT TR0
AND 82.00  ; Pulso bolsa par entrando
SET 54.00  ; Bandera para realizar bolsa 4,8,12 y 16
LD TR0
AND 86.00  ; Rodillos superiores movio OK
SET 55.00  ; Bolsa 4, 8, 12 y 16 en posicion
; rung 10
LD OLD_S6  ; Salida decodificador - Bolsa 6
AND 80.00
OUT TR0
ANDNOT H10.00  ; Habilitacion de Euro Pallet
MOV(021) D505 D1008  ; Bolsa 6
LD TR0
AND H10.00  ; Habilitacion de Euro Pallet
MOV(021) &2 D1008
; rung 11
LD OLD_S7  ; Salida decodificador - Bolsa 7
AND 80.00
MOV(021) D506 D1007
; rung 12
LD OLD_S8  ; Salida decodificador - Bolsa 8
AND 80.00
OUT TR0
ANDNOT H10.00  ; Habilitacion de Euro Pallet
MOV(021) D507 D1008  ; Bolsa 8  // Original valor &8
LD TR0
AND H10.00  ; Habilitacion de Euro Pallet
MOV(021) &2 D1008  // Original valor &8
; rung 13: Muevo pala en Modo normal y Euro
LD OLD_S8  ; Salida decodificador - Bolsa 8
OUT TR0
AND 82.00  ; Pulso bolsa par entrando
SET 54.00  ; Bandera para realizar bolsa 4,8,12 y 16
LD TR0
AND 86.00  ; Rodillos superiores movio OK
SET 55.00  ; Bolsa 4, 8, 12 y 16 en posicion

